(* IEC 61131-3 sources: RAG_PLC/data/result/test/002, 2 files *)

(* ---- wrapped.st ---- *)
(* =========================================================
   Generated by PLC-Eval Benchmark Wrapper
   ========================================================= *)

FUNCTION_BLOCK LLM_Wrapper_FB
VAR_INPUT
    X : REAL;
    T : REAL;
    U : REAL;
END_VAR

VAR
    tmp : REAL;
END_VAR

tmp := X - T;
CAUCHY := 0.318309886183791 * U / (U * U + tmp * tmp);
END_FUNCTION_BLOCK

PROGRAM Auto_Proxy_Prg
  VAR
    instance : LLM_Wrapper_FB;
  END_VAR

  instance();
END_PROGRAM

CONFIGURATION Config0
  RESOURCE Res0 ON PLC
    TASK TaskMain(INTERVAL := T#20ms, PRIORITY := 0);
    PROGRAM Inst0 WITH TaskMain : Auto_Proxy_Prg;
  END_RESOURCE
END_CONFIGURATION

(* ---- raw_code.st ---- *)
VAR_INPUT
    X : REAL;
    T : REAL;
    U : REAL;
END_VAR

VAR
    tmp : REAL;
END_VAR

tmp := X - T;
CAUCHY := 0.318309886183791 * U / (U * U + tmp * tmp);
